// TIA Portal V20 export
// export: Created 2026-07-10T11:12:28.3382873Z, ExportSetting WithDefaults, DisplayName Totally Integrated Automation Portal, DisplayVersion V20, DisplayName TIA Portal Openness, DisplayVersion V20, DisplayName TIA Portal Version Control Interface, DisplayVersion V20, DisplayName STEP 7 Professional, DisplayVersion V20, DisplayName STEP 7 Safety, DisplayVersion V20, DisplayName WinCC Basic/Comfort/Advanced, DisplayVersion V20, DisplayName WinCC Unified, DisplayVersion V20
DATA_BLOCK "Config"   // DB20
{ S7_Optimized_Access := 'FALSE' }
VERSION : 0.1
// stored: AutoNumber false, DBAccessibleFromOPCUA true, IsOnlyStoredInLoadMemory false, IsWriteProtectedInAS false
   VAR
      DateTime : DTL := DTL#2024-10-30-11:20:02.078798;
      HMI_ResetWaterCounter : Bool := FALSE;
      HMI_ResetPositionDamper1 : Bool := FALSE;
      HMI_ResetPositionDamper2 : Bool := FALSE;
      HMI_StartAdjustDamper1 : Bool := FALSE;
      HMI_StartAdjustDamper2 : Bool := FALSE;
      HMI_StopAdjustDamper1 : Bool := FALSE;
      HMI_StopAdjustDamper2 : Bool := FALSE;
      HMI_WeightToZero : Bool := FALSE;
      WaterPulseDuble : Bool;
      DiOxydeDosing : DWord;
   END_VAR
BEGIN
END_DATA_BLOCK
